LIN {X 0,Y 29.537,Z 468.386,A -85,B 0,C 180,E1 -30358.417,E2 -30358.417} C_VEL
LIN {X 0,Y 37.238,Z 465.919,A -85,B 0,C 180,E1 -30379.019,E2 -30379.019} C_VEL
LIN {X 0,Y 45.145,Z 462.963,A -85,B 0,C 180,E1 -30388.895,E2 -30388.895} C_VEL
LIN {X 0,Y 53.962,Z 458.972,A -85,B 0,C 180,E1 -30395.737,E2 -30395.737} C_VEL
LIN {X 0,Y 63.27,Z 453.84,A -85,B 0,C 180,E1 -30400.756,E2 -30400.756} C_VEL
LIN {X 0,Y 68.067,Z 450.884,A -85,B 0,C 180,E1 -30402.76,E2 -30402.76} C_VEL
LIN {X 0,Y 69.528,Z 449.714,A -85,B 0,C 180,E1 -30403.794,E2 -30403.794} C_VEL
LIN {X 0,Y 71.166,Z 448.225,A -85,B 0,C 180,E1 -30405.706,E2 -30405.706} C_VEL
LIN {X 0,Y 72.173,Z 446.933,A -85,B 0,C 180,E1 -30408.767,E2 -30408.767} C_VEL
LIN {X 0,Y 73.195,Z 445.37,A -85,B 0,C 180,E1 -30414.487,E2 -30414.487} C_VEL
LIN {X 0,Y 73.985,Z 444.333,A -85,B 0,C 180,E1 -30419.997,E2 -30419.997} C_VEL
LIN {X 0,Y 72.877,Z 445.263,A -85,B 0,C 180,E1 -30426.742,E2 -30426.742} C_VEL
LIN {X 0,Y 72.114,Z 446.434,A -85,B 0,C 180,E1 -30432.95,E2 -30432.95} C_VEL
LIN {X 0,Y 71.623,Z 447.495,A -85,B 0,C 180,E1 -30437.117,E2 -30437.117} C_VEL
LIN {X 0,Y 70.158,Z 450.002,A -85,B 0,C 180,E1 -30443.618,E2 -30443.618} C_VEL
LIN {X 0,Y 69.177,Z 451.42,A -85,B 0,C 180,E1 -30447.198,E2 -30447.198} C_VEL
LIN {X 0,Y 67.129,Z 454.155,A -85,B 0,C 180,E1 -30453.118,E2 -30453.118} C_VEL
LIN {X 0,Y 63.089,Z 458.862,A -85,B 0,C 180,E1 -30464.284,E2 -30464.284} C_VEL
LIN {X 0,Y 61.528,Z 462.068,A -85,B 0,C 180,E1 -30475.172,E2 -30475.172} C_VEL
LIN {X 0,Y 62.195,Z 464.077,A -85,B 0,C 180,E1 -30484.679,E2 -30484.679} C_VEL
LIN {X 0,Y 66.696,Z 465.871,A -85,B 0,C 180,E1 -30497.834,E2 -30497.834} C_VEL
LIN {X 0,Y 70.831,Z 466.309,A -85,B 0,C 180,E1 -30504.306,E2 -30504.306} C_VEL
LIN {X 0,Y 76.029,Z 466.308,A -85,B 0,C 180,E1 -30510,E2 -30510} C_VEL
LIN {X 0,Y 70.658,Z 466.289,A -85,B 0,C 180,E1 -30515.957,E2 -30515.957} C_VEL
LIN {X 0,Y 65.425,Z 465.602,A -85,B 0,C 180,E1 -30524.822,E2 -30524.822} C_VEL
LIN {X 0,Y 61.957,Z 463.722,A -85,B 0,C 180,E1 -30536.983,E2 -30536.983} C_VEL
LIN {X 0,Y 61.615,Z 461.496,A -85,B 0,C 180,E1 -30547.025,E2 -30547.025} C_VEL
LIN {X 0,Y 64.008,Z 457.653,A -85,B 0,C 180,E1 -30558.797,E2 -30558.797} C_VEL
LIN {X 0,Y 67.116,Z 454.156,A -85,B 0,C 180,E1 -30566.899,E2 -30566.899} C_VEL
LIN {X 0,Y 69.146,Z 451.439,A -85,B 0,C 180,E1 -30572.789,E2 -30572.789} C_VEL
LIN {X 0,Y 70.16,Z 450,A -85,B 0,C 180,E1 -30576.383,E2 -30576.383} C_VEL
LIN {X 0,Y 71.626,Z 447.493,A -85,B 0,C 180,E1 -30582.884,E2 -30582.884} C_VEL
LIN {X 0,Y 72.338,Z 446.047,A -85,B 0,C 180,E1 -30588.799,E2 -30588.799} C_VEL
LIN {X 0,Y 73.137,Z 445.023,A -85,B 0,C 180,E1 -30594.489,E2 -30594.489} C_VEL
LIN {X 0,Y 73.978,Z 444.339,A -85,B 0,C 180,E1 -30600.003,E2 -30600.003} C_VEL
LIN {X 0,Y 72.909,Z 445.701,A -85,B 0,C 180,E1 -30606.669,E2 -30606.669} C_VEL
LIN {X 0,Y 71.717,Z 446.81,A -85,B 0,C 180,E1 -30608.793,E2 -30608.793} C_VEL
LIN {X 0,Y 69.209,Z 448.765,A -85,B 0,C 180,E1 -30610.65,E2 -30610.65} C_VEL
LIN {X 0,Y 66.658,Z 450.531,A -85,B 0,C 180,E1 -30611.714,E2 -30611.714} C_VEL
LIN {X 0,Y 56.67,Z 456.213,A -85,B 0,C 180,E1 -30614.615,E2 -30614.615} C_VEL
LIN {X 0,Y 48.206,Z 460.306,A -85,B 0,C 180,E1 -30618.623,E2 -30618.623} C_VEL
LIN {X 0,Y 38.852,Z 463.919,A -85,B 0,C 180,E1 -30625.249,E2 -30625.249} C_VEL
LIN {X 0,Y 33.001,Z 465.722,A -85,B 0,C 180,E1 -30631.585,E2 -30631.585} C_VEL
LIN {X 0,Y 23.518,Z 468.19,A -85,B 0,C 180,E1 -30653.297,E2 -30653.297} C_VEL
LIN {X 0,Y 20.755,Z 468.791,A -85,B 0,C 180,E1 -30670.207,E2 -30670.207} C_VEL
LIN {X 0,Y 20.02,Z 468.957,A -85,B 0,C 180,E1 -30690,E2 -30690} C_VEL
LIN {X 0,Y 20.75,Z 468.791,A -85,B 0,C 180,E1 -30709.798,E2 -30709.798} C_VEL
LIN {X 0,Y 23.516,Z 468.19,A -85,B 0,C 180,E1 -30726.707,E2 -30726.707} C_VEL
LIN {X 0,Y 33.001,Z 465.722,A -85,B 0,C 180,E1 -30748.414,E2 -30748.414} C_VEL
LIN {X 0,Y 41.909,Z 462.767,A -85,B 0,C 180,E1 -30757.268,E2 -30757.268} C_VEL
LIN {X 0,Y 51.448,Z 458.776,A -85,B 0,C 180,E1 -30762.984,E2 -30762.984} C_VEL
LIN {X 0,Y 61.292,Z 453.643,A -85,B 0,C 180,E1 -30767.056,E2 -30767.056} C_VEL
LIN {X 0,Y 64.627,Z 451.724,A -85,B 0,C 180,E1 -30768.16,E2 -30768.16} C_VEL
LIN {X 0,Y 66.396,Z 450.211,A -85,B 0,C 180,E1 -30771.21,E2 -30771.21} C_VEL
LIN {X 0,Y 66.92,Z 449.514,A -85,B 0,C 180,E1 -30773.968,E2 -30773.968} C_VEL
LIN {X 0,Y 67.973,Z 448.389,A -85,B 0,C 180,E1 -30779.997,E2 -30779.997} C_VEL
LIN {X 0,Y 66.952,Z 449.105,A -85,B 0,C 180,E1 -30786.022,E2 -30786.022} C_VEL
LIN {X 0,Y 66.106,Z 450.2,A -85,B 0,C 180,E1 -30792.273,E2 -30792.273} C_VEL
LIN {X 0,Y 65.645,Z 450.873,A -85,B 0,C 180,E1 -30795.518,E2 -30795.518} C_VEL
LIN {X 0,Y 63.814,Z 452.99,A -85,B 0,C 180,E1 -30802.391,E2 -30802.391} C_VEL
LIN {X 0,Y 62.346,Z 454.697,A -85,B 0,C 180,E1 -30806.798,E2 -30806.798} C_VEL
LIN {X 0,Y 60.898,Z 456.088,A -85,B 0,C 180,E1 -30810.59,E2 -30810.59} C_VEL
LIN {X 0,Y 58.175,Z 458.633,A -85,B 0,C 180,E1 -30817.155,E2 -30817.155} C_VEL
LIN {X 0,Y 54.918,Z 462.297,A -85,B 0,C 180,E1 -30830.219,E2 -30830.219} C_VEL
LIN {X 0,Y 54.938,Z 464.7,A -85,B 0,C 180,E1 -30843.562,E2 -30843.562} C_VEL
LIN {X 0,Y 58.199,Z 466.112,A -85,B 0,C 180,E1 -30856.024,E2 -30856.024} C_VEL
LIN {X 0,Y 63.437,Z 466.649,A -85,B 0,C 180,E1 -30865.572,E2 -30865.572} C_VEL
LIN {X 0,Y 66.99,Z 466.557,A -85,B 0,C 180,E1 -30870,E2 -30870} C_VEL
LIN {X 0,Y 62.041,Z 466.552,A -85,B 0,C 180,E1 -30876.504,E2 -30876.504} C_VEL
LIN {X 0,Y 58.047,Z 466.086,A -85,B 0,C 180,E1 -30884.415,E2 -30884.415} C_VEL
LIN {X 0,Y 54.577,Z 463.955,A -85,B 0,C 180,E1 -30901.003,E2 -30901.003} C_VEL
LIN {X 0,Y 55.59,Z 461.219,A -85,B 0,C 180,E1 -30914.049,E2 -30914.049} C_VEL
LIN {X 0,Y 59.422,Z 457.441,A -85,B 0,C 180,E1 -30925.885,E2 -30925.885} C_VEL
LIN {X 0,Y 60.889,Z 456.097,A -85,B 0,C 180,E1 -30929.386,E2 -30929.386} C_VEL
LIN {X 0,Y 62.585,Z 454.409,A -85,B 0,C 180,E1 -30933.943,E2 -30933.943} C_VEL
LIN {X 0,Y 63.819,Z 452.983,A -85,B 0,C 180,E1 -30937.633,E2 -30937.633} C_VEL
LIN {X 0,Y 65.645,Z 450.873,A -85,B 0,C 180,E1 -30944.482,E2 -30944.482} C_VEL
LIN {X 0,Y 66.108,Z 450.198,A -85,B 0,C 180,E1 -30947.727,E2 -30947.727} C_VEL
LIN {X 0,Y 66.983,Z 449.084,A -85,B 0,C 180,E1 -30953.981,E2 -30953.981} C_VEL
LIN {X 0,Y 67.972,Z 448.39,A -85,B 0,C 180,E1 -30960.003,E2 -30960.003} C_VEL
LIN {X 0,Y 66.905,Z 449.524,A -85,B 0,C 180,E1 -30966.033,E2 -30966.033} C_VEL
LIN {X 0,Y 66.365,Z 450.23,A -85,B 0,C 180,E1 -30968.783,E2 -30968.783} C_VEL
LIN {X 0,Y 64.621,Z 451.723,A -85,B 0,C 180,E1 -30971.818,E2 -30971.818} C_VEL
LIN {X 0,Y 56.67,Z 456.213,A -85,B 0,C 180,E1 -30974.615,E2 -30974.615} C_VEL
LIN {X 0,Y 51.48,Z 458.678,A -85,B 0,C 180,E1 -30976.176,E2 -30976.176} C_VEL
LIN {X 0,Y 45.963,Z 460.859,A -85,B 0,C 180,E1 -30976.908,E2 -30976.908} C_VEL
LIN {X 0,Y 34.581,Z 464.34,A -85,B 0,C 180,E1 -30978.179,E2 -30978.179} C_VEL
LIN {X 0,Y 28.14,Z 466.022,A -85,B 0,C 180,E1 -30981.7,E2 -30981.7} C_VEL
LIN {X 0,Y 27.281,Z 466.108,A -85,B 0,C 180,E1 -30982.622,E2 -30982.622} C_VEL
LIN {X 0,Y 18.313,Z 467.993,A -85,B 0,C 180,E1 -30999.866,E2 -30999.866} C_VEL
LIN {X 0,Y 14.258,Z 468.595,A -85,B 0,C 180,E1 -31020.468,E2 -31020.468} C_VEL
LIN {X 0,Y 12.927,Z 468.761,A -85,B 0,C 180,E1 -31050,E2 -31050} C_VEL
LIN {X 0,Y 14.254,Z 468.595,A -85,B 0,C 180,E1 -31079.541,E2 -31079.541} C_VEL
LIN {X 0,Y 18.311,Z 467.993,A -85,B 0,C 180,E1 -31100.14,E2 -31100.14} C_VEL
LIN {X 0,Y 29.89,Z 465.525,A -85,B 0,C 180,E1 -31120.14,E2 -31120.14} C_VEL
LIN {X 0,Y 39.703,Z 462.57,A -85,B 0,C 180,E1 -31126.797,E2 -31126.797} C_VEL
LIN {X 0,Y 49.828,Z 458.579,A -85,B 0,C 180,E1 -31130.862,E2 -31130.862} C_VEL
LIN {X 0,Y 58.98,Z 454.067,A -85,B 0,C 180,E1 -31133.452,E2 -31133.452} C_VEL
LIN {X 0,Y 60.833,Z 452.927,A -85,B 0,C 180,E1 -31135.17,E2 -31135.17} C_VEL
LIN {X 0,Y 61.71,Z 452.194,A -85,B 0,C 180,E1 -31139.996,E2 -31139.996} C_VEL
LIN {X 0,Y 60.542,Z 452.854,A -85,B 0,C 180,E1 -31146.662,E2 -31146.662} C_VEL
LIN {X 0,Y 59.511,Z 453.91,A -85,B 0,C 180,E1 -31153.658,E2 -31153.658} C_VEL
LIN {X 0,Y 58.714,Z 454.7,A -85,B 0,C 180,E1 -31156.748,E2 -31156.748} C_VEL
LIN {X 0,Y 57.062,Z 456.096,A -85,B 0,C 180,E1 -31161.68,E2 -31161.68} C_VEL
LIN {X 0,Y 55.087,Z 457.677,A -85,B 0,C 180,E1 -31166.739,E2 -31166.739} C_VEL
LIN {X 0,Y 51.502,Z 460.296,A -85,B 0,C 180,E1 -31175.039,E2 -31175.039} C_VEL
LIN {X 0,Y 48.357,Z 462.98,A -85,B 0,C 180,E1 -31186.602,E2 -31186.602} C_VEL
LIN {X 0,Y 47.879,Z 465.435,A -85,B 0,C 180,E1 -31203.873,E2 -31203.873} C_VEL
LIN {X 0,Y 50.662,Z 466.474,A -85,B 0,C 180,E1 -31216.164,E2 -31216.164} C_VEL
LIN {X 0,Y 58.079,Z 466.803,A -85,B 0,C 180,E1 -31230,E2 -31230} C_VEL
LIN {X 0,Y 50.671,Z 466.471,A -85,B 0,C 180,E1 -31243.875,E2 -31243.875} C_VEL
LIN {X 0,Y 47.713,Z 465.249,A -85,B 0,C 180,E1 -31257.907,E2 -31257.907} C_VEL
LIN {X 0,Y 48.864,Z 462.525,A -85,B 0,C 180,E1 -31275.983,E2 -31275.983} C_VEL
LIN {X 0,Y 52.643,Z 459.531,A -85,B 0,C 180,E1 -31287.728,E2 -31287.728} C_VEL
LIN {X 0,Y 55.079,Z 457.677,A -85,B 0,C 180,E1 -31293.276,E2 -31293.276} C_VEL
LIN {X 0,Y 57.047,Z 456.104,A -85,B 0,C 180,E1 -31298.314,E2 -31298.314} C_VEL
LIN {X 0,Y 58.718,Z 454.7,A -85,B 0,C 180,E1 -31303.241,E2 -31303.241} C_VEL
LIN {X 0,Y 59.511,Z 453.91,A -85,B 0,C 180,E1 -31306.342,E2 -31306.342} C_VEL
LIN {X 0,Y 60.586,Z 452.83,A -85,B 0,C 180,E1 -31313.342,E2 -31313.342} C_VEL
LIN {X 0,Y 61.705,Z 452.196,A -85,B 0,C 180,E1 -31320.004,E2 -31320.004} C_VEL
LIN {X 0,Y 60.824,Z 452.93,A -85,B 0,C 180,E1 -31324.803,E2 -31324.803} C_VEL
LIN {X 0,Y 58.975,Z 454.067,A -85,B 0,C 180,E1 -31326.522,E2 -31326.522} C_VEL
LIN {X 0,Y 49.827,Z 458.578,A -85,B 0,C 180,E1 -31329.127,E2 -31329.127} C_VEL
LIN {X 0,Y 39.703,Z 462.57,A -85,B 0,C 180,E1 -31333.201,E2 -31333.201} C_VEL
LIN {X 0,Y 29.89,Z 465.525,A -85,B 0,C 180,E1 -31339.86,E2 -31339.86} C_VEL
LIN {X 0,Y 27.281,Z 466.108,A -85,B 0,C 180,E1 -31342.622,E2 -31342.622} C_VEL
LIN {X 0,Y 22.038,Z 467.218,A -85,B 0,C 180,E1 -31348.518,E2 -31348.518} C_VEL
LIN {X 0,Y 16.597,Z 467.977,A -85,B 0,C 180,E1 -31355.318,E2 -31355.318} C_VEL
LIN {X 0,Y 6.948,Z 468.589,A -85,B 0,C 180,E1 -31393.968,E2 -31393.968} C_VEL
LIN {X 0,Y 8.034,Z 468.424,A -85,B 0,C 180,E1 -31458.052,E2 -31458.052} C_VEL
LIN {X 0,Y 14.792,Z 467.797,A -85,B 0,C 180,E1 -31481.849,E2 -31481.849} C_VEL
LIN {X 0,Y 28.275,Z 465.329,A -85,B 0,C 180,E1 -31493.848,E2 -31493.848} C_VEL
LIN {X 0,Y 38.702,Z 462.373,A -85,B 0,C 180,E1 -31497.145,E2 -31497.145} C_VEL
LIN {X 0,Y 49.202,Z 458.382,A -85,B 0,C 180,E1 -31499.101,E2 -31499.101} C_VEL
LIN {X 0,Y 55.269,Z 455.665,A -85,B 0,C 180,E1 -31499.996,E2 -31499.996} C_VEL
LIN {X 0,Y 53.884,Z 456.309,A -85,B 0,C 180,E1 -31507.49,E2 -31507.49} C_VEL
LIN {X 0,Y 51.949,Z 457.614,A -85,B 0,C 180,E1 -31515.694,E2 -31515.694} C_VEL
LIN {X 0,Y 49.383,Z 459.365,A -85,B 0,C 180,E1 -31522.334,E2 -31522.334} C_VEL
LIN {X 0,Y 43.539,Z 462.752,A -85,B 0,C 180,E1 -31536.187,E2 -31536.187} C_VEL
LIN {X 0,Y 41.178,Z 464.415,A -85,B 0,C 180,E1 -31546.946,E2 -31546.946} C_VEL
LIN {X 0,Y 41.721,Z 466.586,A -85,B 0,C 180,E1 -31570.312,E2 -31570.312} C_VEL
LIN {X 0,Y 44.685,Z 467.035,A -85,B 0,C 180,E1 -31580.951,E2 -31580.951} C_VEL
LIN {X 0,Y 49.192,Z 467.048,A -85,B 0,C 180,E1 -31590.093,E2 -31590.093} C_VEL
LIN {X 0,Y 43.306,Z 466.853,A -85,B 0,C 180,E1 -31603.189,E2 -31603.189} C_VEL
LIN {X 0,Y 40.503,Z 465.667,A -85,B 0,C 180,E1 -31621.369,E2 -31621.369} C_VEL
LIN {X 0,Y 42.032,Z 463.674,A -85,B 0,C 180,E1 -31638.031,E2 -31638.031} C_VEL
LIN {X 0,Y 47.417,Z 460.426,A -85,B 0,C 180,E1 -31653.604,E2 -31653.604} C_VEL
LIN {X 0,Y 49.378,Z 459.365,A -85,B 0,C 180,E1 -31657.679,E2 -31657.679} C_VEL
LIN {X 0,Y 51.948,Z 457.614,A -85,B 0,C 180,E1 -31664.306,E2 -31664.306} C_VEL
LIN {X 0,Y 53.914,Z 456.296,A -85,B 0,C 180,E1 -31672.514,E2 -31672.514} C_VEL
LIN {X 0,Y 54.774,Z 455.903,A -85,B 0,C 180,E1 -31680.004,E2 -31680.004} C_VEL
LIN {X 0,Y 45.696,Z 459.913,A -85,B 0,C 180,E1 -31681.454,E2 -31681.454} C_VEL
LIN {X 0,Y 35.217,Z 463.526,A -85,B 0,C 180,E1 -31683.786,E2 -31683.786} C_VEL
LIN {X 0,Y 24.623,Z 466.071,A -85,B 0,C 180,E1 -31688.056,E2 -31688.056} C_VEL
LIN {X 0,Y 14.793,Z 467.797,A -85,B 0,C 180,E1 -31698.157,E2 -31698.157} C_VEL
LIN {X 0,Y 8.799,Z 468.399,A -85,B 0,C 180,E1 -31716.994,E2 -31716.994} C_VEL
LIN {X 0,Y 5.821,Z 468.565,A -85,B 0,C 180,E1 -31770,E2 -31770} C_VEL
LIN {X 0,Y 8.034,Z 468.424,A -85,B 0,C 180,E1 -31818.052,E2 -31818.052} C_VEL
LIN {X 0,Y 12.492,Z 468.128,A -85,B 0,C 180,E1 -31840.243,E2 -31840.243} C_VEL
LIN {X 0,Y 20.85,Z 466.976,A -85,B 0,C 180,E1 -31858.806,E2 -31858.806} C_VEL
LIN {X 0,Y 28.106,Z 465.427,A -85,B 0,C 180,E1 -31865.732,E2 -31865.732} C_VEL
LIN {X 0,Y 33.739,Z 463.872,A -85,B 0,C 180,E1 -31867.674,E2 -31867.674} C_VEL
LIN {X 0,Y 35.625,Z 463.277,A -85,B 0,C 180,E1 -31867.766,E2 -31867.766} C_VEL
LIN {X 0,Y 42.54,Z 460.957,A -85,B 0,C 180,E1 -31867.588,E2 -31867.588} C_VEL
LIN {X 0,Y 46.631,Z 459.52,A -85,B 0,C 180,E1 -31868.664,E2 -31868.664} C_VEL
LIN {X 0,Y 44.004,Z 460.765,A -85,B 0,C 180,E1 -31876.609,E2 -31876.609} C_VEL
LIN {X 0,Y 39.282,Z 462.977,A -85,B 0,C 180,E1 -31886.548,E2 -31886.548} C_VEL
LIN {X 0,Y 35.585,Z 464.643,A -85,B 0,C 180,E1 -31897.816,E2 -31897.816} C_VEL
LIN {X 0,Y 33.83,Z 466.821,A -85,B 0,C 180,E1 -31925.45,E2 -31925.45} C_VEL
LIN {X 0,Y 36.193,Z 467.273,A -85,B 0,C 180,E1 -31938.803,E2 -31938.803} C_VEL
LIN {X 0,Y 40.473,Z 467.288,A -85,B 0,C 180,E1 -31950,E2 -31950} C_VEL
LIN {X 0,Y 35.95,Z 467.235,A -85,B 0,C 180,E1 -31962.218,E2 -31962.218} C_VEL
LIN {X 0,Y 33.449,Z 466.338,A -85,B 0,C 180,E1 -31982.825,E2 -31982.825} C_VEL
LIN {X 0,Y 36.082,Z 464.367,A -85,B 0,C 180,E1 -32004.251,E2 -32004.251} C_VEL
LIN {X 0,Y 39.28,Z 462.977,A -85,B 0,C 180,E1 -32013.457,E2 -32013.457} C_VEL
LIN {X 0,Y 44.002,Z 460.765,A -85,B 0,C 180,E1 -32023.396,E2 -32023.396} C_VEL
LIN {X 0,Y 46.668,Z 459.504,A -85,B 0,C 180,E1 -32031.343,E2 -32031.343} C_VEL
LIN {X 0,Y 42.541,Z 460.957,A -85,B 0,C 180,E1 -32032.409,E2 -32032.409} C_VEL
LIN {X 0,Y 35.466,Z 463.329,A -85,B 0,C 180,E1 -32032.229,E2 -32032.229} C_VEL
LIN {X 0,Y 28.408,Z 465.133,A -85,B 0,C 180,E1 -32031.724,E2 -32031.724} C_VEL
LIN {X 0,Y 14.282,Z 467.6,A -85,B 0,C 180,E1 -32029.783,E2 -32029.783} C_VEL
LIN {X 0,Y 7.264,Z 468.202,A -85,B 0,C 180,E1 -32025.354,E2 -32025.354} C_VEL
LIN {X 0,Y 1.291,Z 468.369,A -85,B 0,C 180,E1 -31950,E2 -31950} C_VEL
LIN {X 0,Y 7.265,Z 468.202,A -85,B 0,C 180,E1 -31874.672,E2 -31874.672} C_VEL
LIN {X 0,Y 14.283,Z 467.6,A -85,B 0,C 180,E1 -31870.223,E2 -31870.223} C_VEL
LIN {X 0,Y 28.408,Z 465.133,A -85,B 0,C 180,E1 -31868.275,E2 -31868.275} C_VEL
LIN {X 0,Y 35.625,Z 463.277,A -85,B 0,C 180,E1 -31867.766,E2 -31867.766} C_VEL
LIN {X 0,Y 34.694,Z 463.541,A -85,B 0,C 180,E1 -31869.731,E2 -31869.731} C_VEL
LIN {X 0,Y 28.519,Z 465.192,A -85,B 0,C 180,E1 -31875.36,E2 -31875.36} C_VEL
LIN {X 0,Y 18.26,Z 467.217,A -85,B 0,C 180,E1 -31888.584,E2 -31888.584} C_VEL
LIN {X 0,Y 11.548,Z 467.981,A -85,B 0,C 180,E1 -31910.563,E2 -31910.563} C_VEL
LIN {X 0,Y 9.809,Z 468.067,A -85,B 0,C 180,E1 -31923.151,E2 -31923.151} C_VEL
LIN {X 0,Y 8.392,Z 468.173,A -85,B 0,C 180,E1 -31950,E2 -31950} C_VEL
LIN {X 0,Y 11.388,Z 468.005,A -85,B 0,C 180,E1 -31988.109,E2 -31988.109} C_VEL
LIN {X 0,Y 17.061,Z 467.403,A -85,B 0,C 180,E1 -32005.471,E2 -32005.471} C_VEL
LIN {X 0,Y 30.262,Z 464.936,A -85,B 0,C 180,E1 -32018.273,E2 -32018.273} C_VEL
LIN {X 0,Y 32.574,Z 464.394,A -85,B 0,C 180,E1 -32017.625,E2 -32017.625} C_VEL
LIN {X 0,Y 26.514,Z 466.87,A -85,B 0,C 180,E1 -31987.34,E2 -31987.34} C_VEL
LIN {X 0,Y 28.619,Z 467.599,A -85,B 0,C 180,E1 -31960.847,E2 -31960.847} C_VEL
LIN {X 0,Y 31.797,Z 467.528,A -85,B 0,C 180,E1 -31950,E2 -31950} C_VEL
LIN {X 0,Y 27.885,Z 467.508,A -85,B 0,C 180,E1 -31935.402,E2 -31935.402} C_VEL
LIN {X 0,Y 26.515,Z 466.87,A -85,B 0,C 180,E1 -31912.657,E2 -31912.657} C_VEL
LIN {X 0,Y 32.58,Z 464.392,A -85,B 0,C 180,E1 -31882.374,E2 -31882.374} C_VEL
LIN {X 0,Y 30.262,Z 464.936,A -85,B 0,C 180,E1 -31881.727,E2 -31881.727} C_VEL
LIN {X 0,Y 17.062,Z 467.403,A -85,B 0,C 180,E1 -31894.532,E2 -31894.532} C_VEL
LIN {X 0,Y 9.809,Z 468.067,A -85,B 0,C 180,E1 -31923.151,E2 -31923.151} C_VEL
LIN {X 0,Y 9.132,Z 468.157,A -85,B 0,C 180,E1 -31947.37,E2 -31947.37} C_VEL
LIN {X 0,Y 11.055,Z 468.115,A -85,B 0,C 180,E1 -31968.015,E2 -31968.015} C_VEL
LIN {X 0,Y 14.95,Z 467.9,A -85,B 0,C 180,E1 -31979.812,E2 -31979.812} C_VEL
LIN {X 0,Y 17.719,Z 467.686,A -85,B 0,C 180,E1 -31980.845,E2 -31980.845} C_VEL
LIN {X 0,Y 19.235,Z 467.609,A -85,B 0,C 180,E1 -31978.569,E2 -31978.569} C_VEL
LIN {X 0,Y 19.453,Z 467.621,A -85,B 0,C 180,E1 -31977.18,E2 -31977.18} C_VEL
LIN {X 0,Y 23.196,Z 467.765,A -85,B 0,C 180,E1 -31950,E2 -31950} C_VEL
LIN {X 0,Y 19.451,Z 467.621,A -85,B 0,C 180,E1 -31922.824,E2 -31922.824} C_VEL
LIN {X 0,Y 17.546,Z 467.809,A -85,B 0,C 180,E1 -31926.388,E2 -31926.388} C_VEL
LIN {X 0,Y 15.509,Z 467.977,A -85,B 0,C 180,E1 -31950,E2 -31950} C_VEL
LIN {X 0,Y 17.544,Z 467.809,A -85,B 0,C 180,E1 -31973.615,E2 -31973.615} C_VEL
LIN {X 0,Y 19.453,Z 467.621,A -85,B 0,C 180,E1 -31977.18,E2 -31977.18} C_VEL
LIN {X 0,Y 21.37,Z 469.614,A -85,B 0,C 180,E1 -31980.027,E2 -31980.027} C_VEL
LIN {X 0,Y 21.37,Z 600,A -85,B 0,C 180,E1 -31980.027,E2 -31980.027} C_VEL
LIN {X 0,Y 21.37,Z 600,A -85,B 0,C 180,E1 -31980.027,E2 -31980.027}

QRS_NEXT_CUT()

QRS_NEXT()
QRS_HOME()

END
